FUNCTION_BLOCK ABSTRACT AwaitableError IMPLEMENTS Callback
VAR_INPUT
	errorName: STRING;
	errorMessage: STRING(255);
	onErrorStep: UDINT := 0;
END_VAR
VAR_OUTPUT
END_VAR
VAR
END_VAR

(* This is method get's exectued by the framework when the callback is triggered.
 It returns a step number which might be used together with Await to jump to a certain chain step
 after the callback code has been executed.*)
METHOD execute : UDINT
execute := onErrorStep;
END_METHOD

METHOD getMessage : String(255)
VAR_INPUT
END_VAR
getMessage := errorMessage;
END_METHOD

METHOD getName : String
VAR_INPUT
END_VAR
getName := errorName;
END_METHOD

END_FUNCTION_BLOCK

(* stored: Version 1.1.0.1, ProductVersion 3.1.4024.12
   POU AwaitableError: Id {f013d3f3-35b1-42e4-9cd5-becbda020fda}, SpecialFunc None
   Method execute: Id {625e57cf-8c9e-4b1e-9d42-9ab0ea12969b}
   Method getMessage: Id {e9dd875b-0c3c-42b2-a358-703b11eccf52}
   Method getName: Id {f5227696-795c-45c3-b511-c7a28392c6d7} *)
